FUNCTION_BLOCK F_ATAN2 (* principal arc tan of Y/X *)
  (* Standard: 61131-3; Classification: standard function of two numeric variables; Description: Copyright (c) 2013 TU Wien ACIN, Patrick Aigner, HR Agrartechnik GmbH This program and the accompanying materials are made available under the terms of the Eclipse Public License 2.0 which is available at https://www.eclipse.org/legal/epl-2.0/ SPDX-License-Identifier: EPL-2.0 Some portions generated by Gemini CLI *)
  (* Version 1.0, 2026-02-01, Franz H??pfinger, HR Agrartechnik GmbH, copy from F_ATAN an make initial Version *)
  PACKAGE iec61131::numerical;
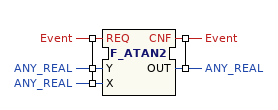
  EVENT_INPUT
    REQ WITH Y, X; (* Service Request *)
  END_EVENT
  EVENT_OUTPUT
    CNF WITH OUT; (* Confirmation of Requested Service *)
  END_EVENT
  VAR_INPUT
    Y : ANY_REAL; (* Ordinate *)
    X : ANY_REAL; (* Abscissa *)
  END_VAR
  VAR_OUTPUT
    OUT : ANY_REAL; (* Result *)
  END_VAR
  EC_STATES
    REQ : REQ -> CNF;
  END_STATES
  ALGORITHM REQ IN ST:
OUT := ATAN2(X, Y);
  END_ALGORITHM
END_FUNCTION_BLOCK
